(* PLC project Unnamed, Unknown Unnamed 1 *)
(* stored: creationDateTime 2024-09-03T16:04:08, modificationDateTime 2025-03-21T02:56:36 *)

PROGRAM irrigation_ST
  VAR
    SoilMoisture AT %IW0.0 : INT;  (* Soil moisture input from Modbus *)
  END_VAR
  VAR
    SoilMoistureMin : INT := 350;  (* Soil moisture below this -> needs watering *)
    SoilMoistureMax : INT := 600;  (* oil moisture above this -> well hydrated *)
  END_VAR
  VAR
    Temperature AT %IW0.1 : INT;  (* Temperature input from Modbus *)
  END_VAR
  VAR
    TempMin : INT := 10;  (* Temperature lower bound *)
    TempMax : INT := 35;  (* Temperature upper bound *)
  END_VAR
  VAR
    Humidity AT %IW0.2 : INT;  (* Humidity input from Modbus *)
  END_VAR
  VAR
    HumidityMin : INT := 40;  (* Humidity lower bound *)
    HumidityMax : INT := 80;  (* Humidity upper bound *)
  END_VAR
  VAR
    WaterFlow AT %IW0.3 : INT;  (* Water flow input from Modbus *)
  END_VAR
  VAR
    FlowMin : INT := 300;  (* Water flow lower bound *)
    FlowMax : INT := 800;  (* Water flow upper bound *)
  END_VAR
  VAR
    Pressure AT %IW0.4 : INT;  (* Pressure input from Modbus *)
  END_VAR
  VAR
    PressureMin : INT := 60;  (* Pressure lower bound *)
    PressureMax : INT := 100;  (* Pressure upper bound *)
    PumpReady : BOOL := FALSE;  (* internal marker for valve open status *)
  END_VAR
  VAR
    PumpControl AT %QX0.0 : BOOL;  (* Output to control the pump *)
  END_VAR
  VAR
    ValveReady : BOOL := FALSE;  (* internal marker for pump on status *)
  END_VAR
  VAR
    ValveControl AT %QX0.1 : BOOL;  (* Output to control the valve *)
  END_VAR

            (* 1) Check if we need irrigation:
      - Soil moisture < min
      - Temperature between TempMin and TempMax
      - Humidity between HumidityMin and HumidityMax
   If we need irrigation, we begin the sequence:
      - Open valve
      - Wait for valve to be considered "open" (here simplified by a marker or short dwell)
      - Turn on pump
*)

IF (SoilMoisture < SoilMoistureMin) 
   AND (Temperature >= TempMin AND Temperature <= TempMax)
   AND (Humidity >= HumidityMin AND Humidity <= HumidityMax) THEN
      ValveControl := TRUE;
      PumpControl := TRUE;


ELSE
   (*
      If conditions are out of range or we have enough moisture:
      - Turn off the pump (PumpReady = FALSE)
      - Once the pump is confirmed off, close the valve
   *)
    PumpControl := FALSE;
    ValveControl := FALSE;
END_IF;
          
END_PROGRAM

CONFIGURATION Config0
  RESOURCE Res0 ON PLC
    TASK task0(INTERVAL := T#20ms, PRIORITY := 0);
    PROGRAM instance0 WITH task0 : irrigation_ST;
  END_RESOURCE
END_CONFIGURATION
